// Mitsubishi GX Works2 project: unity   PLC: Q03UD

PROGRAM CV2
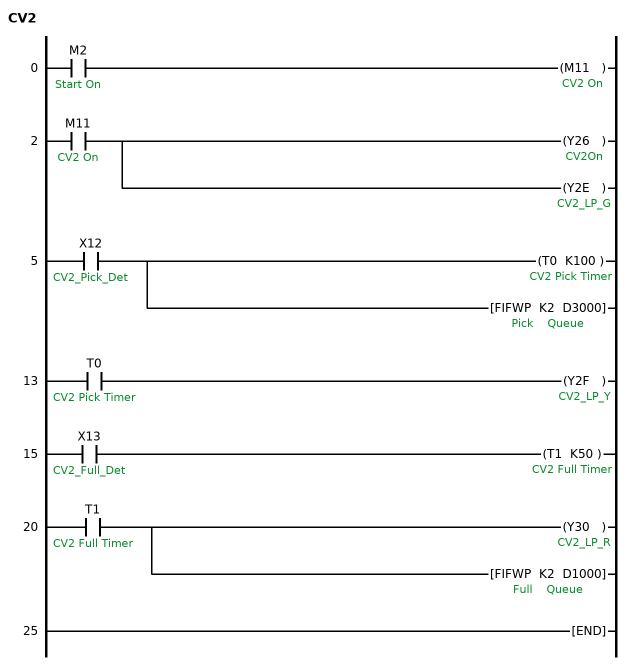
0     LD      M2  ; Start On
      OUT     M11  ; CV2 On
2     LD      M11  ; CV2 On
      OUT     Y26  ; CV2On
      OUT     Y2E  ; CV2_LP_G
5     LD      X12  ; CV2_Pick_Det
      OUT     T0 K100  ; CV2 Pick Timer
      FIFWP   K2 D3000  ; Pick    Queue
13    LD      T0  ; CV2 Pick Timer
      OUT     Y2F  ; CV2_LP_Y
15    LD      X13  ; CV2_Full_Det
      OUT     T1 K50  ; CV2 Full Timer
20    LD      T1  ; CV2 Full Timer
      OUT     Y30  ; CV2_LP_R
      FIFWP   K2 D1000  ; Full    Queue
25    END
END_PROGRAM

PROGRAM CV3
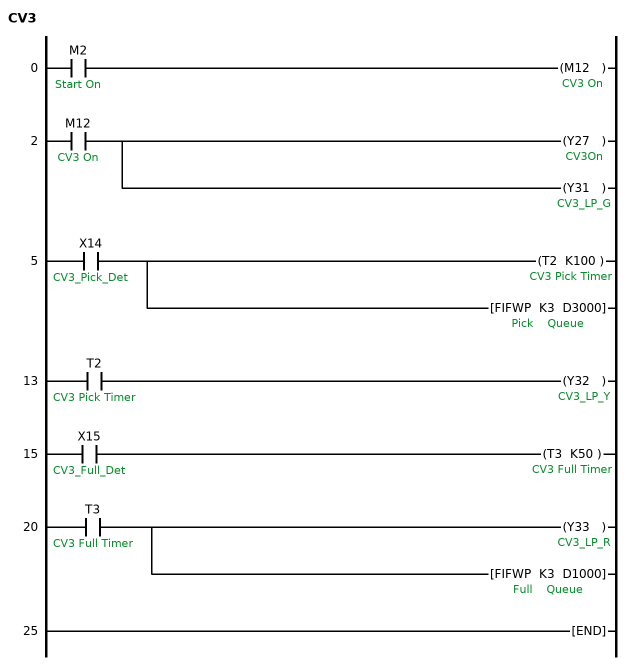
0     LD      M2  ; Start On
      OUT     M12  ; CV3 On
2     LD      M12  ; CV3 On
      OUT     Y27  ; CV3On
      OUT     Y31  ; CV3_LP_G
5     LD      X14  ; CV3_Pick_Det
      OUT     T2 K100  ; CV3 Pick Timer
      FIFWP   K3 D3000  ; Pick    Queue
13    LD      T2  ; CV3 Pick Timer
      OUT     Y32  ; CV3_LP_Y
15    LD      X15  ; CV3_Full_Det
      OUT     T3 K50  ; CV3 Full Timer
20    LD      T3  ; CV3 Full Timer
      OUT     Y33  ; CV3_LP_R
      FIFWP   K3 D1000  ; Full    Queue
25    END
END_PROGRAM

PROGRAM CV4
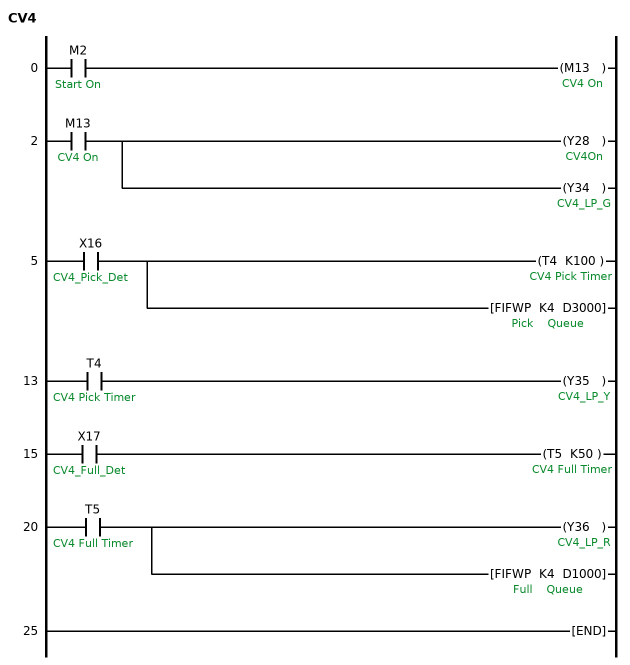
0     LD      M2  ; Start On
      OUT     M13  ; CV4 On
2     LD      M13  ; CV4 On
      OUT     Y28  ; CV4On
      OUT     Y34  ; CV4_LP_G
5     LD      X16  ; CV4_Pick_Det
      OUT     T4 K100  ; CV4 Pick Timer
      FIFWP   K4 D3000  ; Pick    Queue
13    LD      T4  ; CV4 Pick Timer
      OUT     Y35  ; CV4_LP_Y
15    LD      X17  ; CV4_Full_Det
      OUT     T5 K50  ; CV4 Full Timer
20    LD      T5  ; CV4 Full Timer
      OUT     Y36  ; CV4_LP_R
      FIFWP   K4 D1000  ; Full    Queue
25    END
END_PROGRAM

PROGRAM CV5
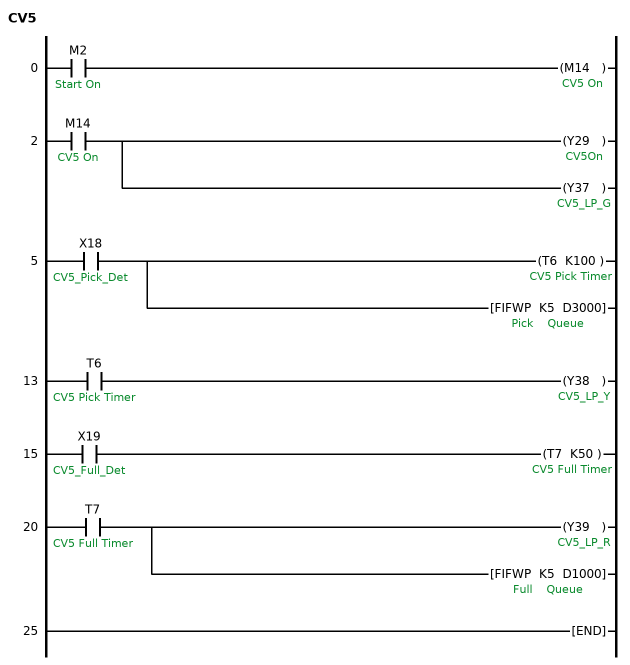
0     LD      M2  ; Start On
      OUT     M14  ; CV5 On
2     LD      M14  ; CV5 On
      OUT     Y29  ; CV5On
      OUT     Y37  ; CV5_LP_G
5     LD      X18  ; CV5_Pick_Det
      OUT     T6 K100  ; CV5 Pick Timer
      FIFWP   K5 D3000  ; Pick    Queue
13    LD      T6  ; CV5 Pick Timer
      OUT     Y38  ; CV5_LP_Y
15    LD      X19  ; CV5_Full_Det
      OUT     T7 K50  ; CV5 Full Timer
20    LD      T7  ; CV5 Full Timer
      OUT     Y39  ; CV5_LP_R
      FIFWP   K5 D1000  ; Full    Queue
25    END
END_PROGRAM

PROGRAM OpPanel
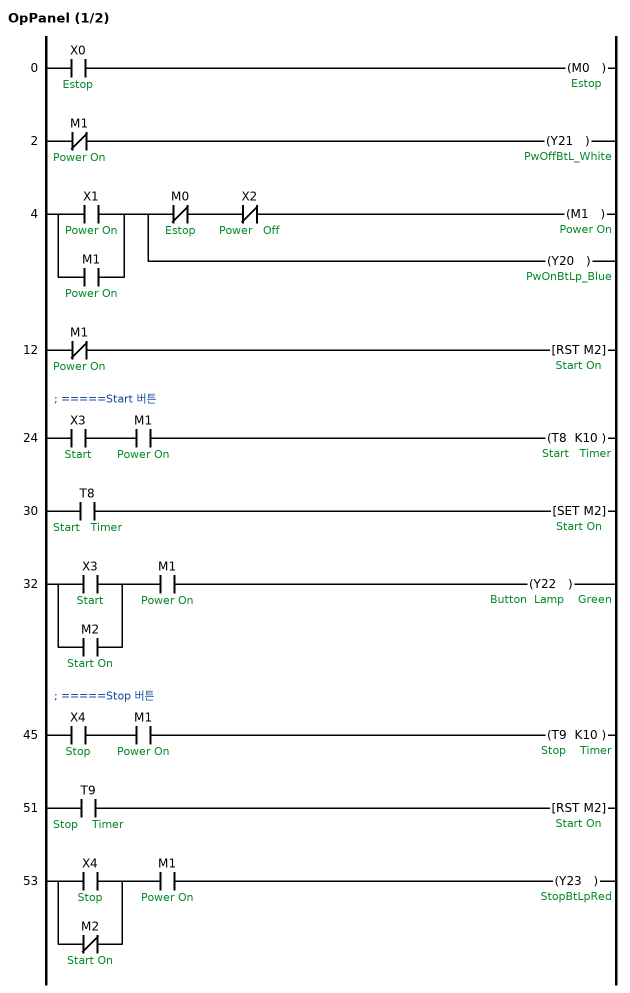
0     LD      X0  ; Estop
      OUT     M0  ; Estop
2     LDI     M1  ; Power On
      OUT     Y21  ; PwOffBtL_White
4     LD      X1  ; Power On
      OR      M1  ; Power On
      MPS
      ANI     M0  ; Estop
      ANI     X2  ; Power   Off
      OUT     M1  ; Power On
      MPP
      OUT     Y20  ; PwOnBtLp_Blue
12    LDI     M1  ; Power On
      RST     M2  ; Start On
; =====Start 버튼
24    LD      X3  ; Start
      AND     M1  ; Power On
      OUT     T8 K10  ; Start   Timer
30    LD      T8  ; Start   Timer
      SET     M2  ; Start On
32    LD      X3  ; Start
      OR      M2  ; Start On
      AND     M1  ; Power On
      OUT     Y22  ; Button  Lamp    Green
; =====Stop 버튼
45    LD      X4  ; Stop
      AND     M1  ; Power On
      OUT     T9 K10  ; Stop    Timer
51    LD      T9  ; Stop    Timer
      RST     M2  ; Start On
53    LD      X4  ; Stop
      ORI     M2  ; Start On
      AND     M1  ; Power On
      OUT     Y23  ; StopBtLpRed
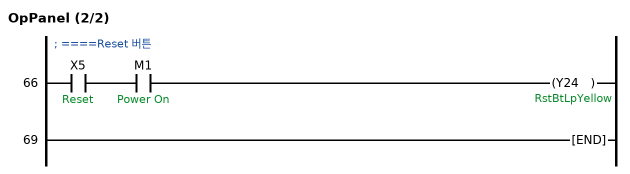
; ====Reset 버튼
66    LD      X5  ; Reset
      AND     M1  ; Power On
      OUT     Y24  ; RstBtLpYellow
69    END
END_PROGRAM

PROGRAM Machin
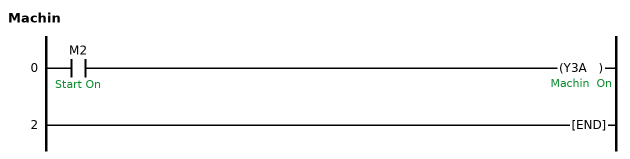
0     LD      M2  ; Start On
      OUT     Y3A  ; Machin  On
2     END
END_PROGRAM

PROGRAM CV1
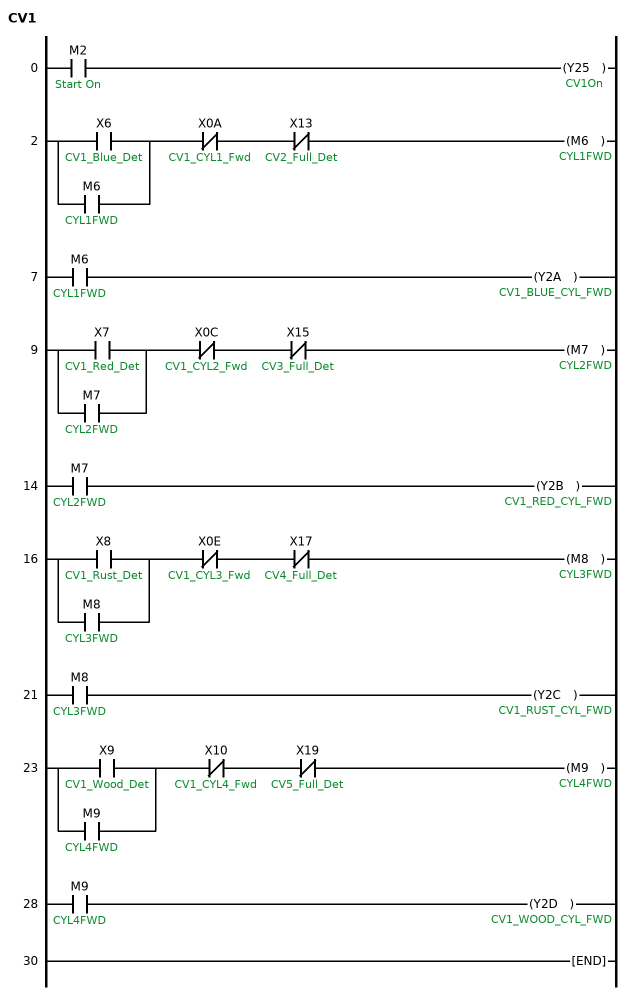
0     LD      M2  ; Start On
      OUT     Y25  ; CV1On
2     LD      X6  ; CV1_Blue_Det
      OR      M6  ; CYL1FWD
      ANI     X0A  ; CV1_CYL1_Fwd
      ANI     X13  ; CV2_Full_Det
      OUT     M6  ; CYL1FWD
7     LD      M6  ; CYL1FWD
      OUT     Y2A  ; CV1_BLUE_CYL_FWD
9     LD      X7  ; CV1_Red_Det
      OR      M7  ; CYL2FWD
      ANI     X0C  ; CV1_CYL2_Fwd
      ANI     X15  ; CV3_Full_Det
      OUT     M7  ; CYL2FWD
14    LD      M7  ; CYL2FWD
      OUT     Y2B  ; CV1_RED_CYL_FWD
16    LD      X8  ; CV1_Rust_Det
      OR      M8  ; CYL3FWD
      ANI     X0E  ; CV1_CYL3_Fwd
      ANI     X17  ; CV4_Full_Det
      OUT     M8  ; CYL3FWD
21    LD      M8  ; CYL3FWD
      OUT     Y2C  ; CV1_RUST_CYL_FWD
23    LD      X9  ; CV1_Wood_Det
      OR      M9  ; CYL4FWD
      ANI     X10  ; CV1_CYL4_Fwd
      ANI     X19  ; CV5_Full_Det
      OUT     M9  ; CYL4FWD
28    LD      M9  ; CYL4FWD
      OUT     Y2D  ; CV1_WOOD_CYL_FWD
30    END
END_PROGRAM

PROGRAM Manager
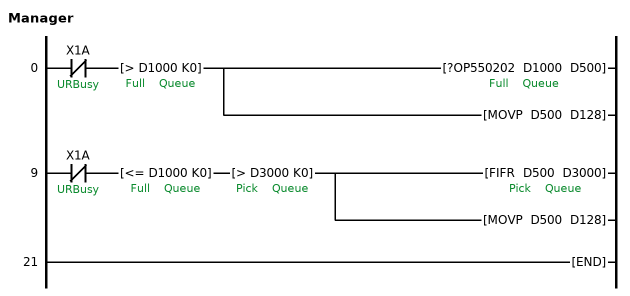
0     LDI     X1A  ; URBusy
      AND>    D1000 K0  ; Full    Queue
      ?OP550202 D1000 D500
      MOVP    D500 D128
9     LDI     X1A  ; URBusy
      AND<=   D1000 K0  ; Full    Queue
      AND>    D3000 K0  ; Pick    Queue
      FIFR    D500 D3000
      MOVP    D500 D128
21    END
END_PROGRAM

// device comments not shown above
X0B  ; CV1_CYL1_Bwd
X0D  ; CV1_CYL2_Bwd
X0F  ; CV1_CYL2_Bwd
X11  ; CV1_CYL4_Bwd
X1B  ; Axis0 Moving
T10  ; CV2     Pick OffTimer
T11  ; CV3     Pick OffTimer
T12  ; CV4     Pick OffTimer
T13  ; CV5     Pick OffTimer
T14  ; CV5     Empty   Timer
T15  ; CV4     Empty   Timer
T16  ; CV3     Empty   Timer
T18  ; CV2     Empty   Timer
M3  ; Power   Off
M4  ; Stop On
M10  ; CV1 On
M15  ; Robot   ready
D501  ; 컨베이어 작업 순서
D1001  ; Full    Queue   Size
D2000  ; Delay   Queue
D3001  ; Pick    Queue   Size
D3002  ; 2번째
D3003  ; 3번째
D3004  ; 4번째
